PROGRAM Vision
VAR
  trigVisionOk    : R_TRIG;	

//System_Bit
	Always_ON	:	BOOL	:=TRUE	;//상시 ON 
	Always_OFF	:	BOOL	:=FALSE	;//상시 OFF
	
	
	TON_1: TON;
	Time_Data_1: LREAL ;
	
	DATA : LREAL;
	

	CCTV: TON;
	Work_End_Position_Set: BOOL;
	GVL_Vision_ON_Delay_Time: INT;
	test005: BOOL;
	Vision_Delay: BOOL;
	Vision_Delay_TM: TON;
	test01: BOOL;
	Vision_NG_Timer: TON;
	Vision_OFF_Dealy: TON;
	TON_0: TON;
END_VAR
VAR // added by the converter: edge detectors and wires of the graphical bodies
    _rt1, _rt2, _rt3, _rt4, _rt5 : R_TRIG;
    _w1, _w2 : BOOL;
END_VAR

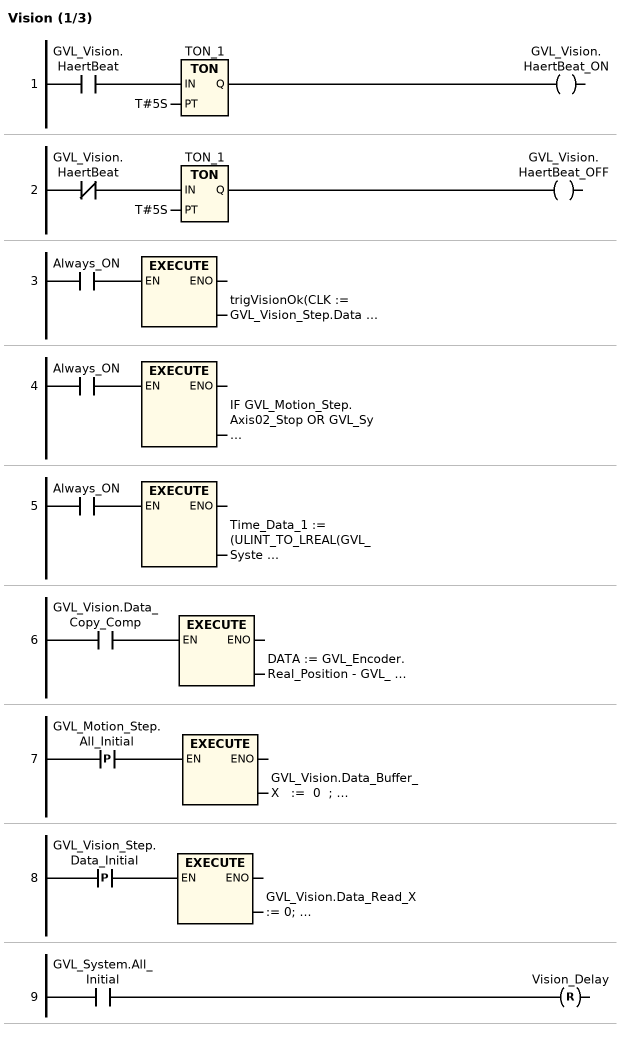
// NETWORK 1
TON_1(IN := GVL_Vision.HaertBeat, PT := T#5S); // TON
GVL_Vision.HaertBeat_ON := TON_1.Q;

// NETWORK 2
TON_1(IN := NOT GVL_Vision.HaertBeat, PT := T#5S); // TON
GVL_Vision.HaertBeat_OFF := TON_1.Q;

// NETWORK 3
IF Always_ON THEN
    trigVisionOk(CLK := GVL_Vision_Step.Data_Initial);
    
    IF trigVisionOk.Q OR GVL_System.All_Initial THEN
    	GVL_Vision.Data_Read_X	:=	0;
    	GVL_Vision.Data_Read_Y	:=	0;
    	GVL_Vision.Data_Read_R	:=	0;
    	GVL_Vision.Vision_OK	:=	FALSE;
    	GVL_Vision.Vision_NG	:=	FALSE;
    END_IF
END_IF

// NETWORK 4
IF Always_ON THEN
    IF GVL_Motion_Step.Axis02_Stop OR GVL_System.All_Initial THEN
    	GVL_Vision.Average_Speed := 0;
    	GVL_Vision.TotalSpeed := 0;
    	GVL_Vision.FrameCount := 0;
    	GVL_Vision.Get_Frame := 0;
    	DATA := 0;
    END_IF
END_IF

// NETWORK 5
IF Always_ON THEN
    
    Time_Data_1 := (ULINT_TO_LREAL(GVL_System.Time_Data) * 1E-7);
    
    IF GVL_Vision.Data_Copy_Comp THEN
    	 GVL_Vision.Moving_Time := Time_Data_1 - GVL_Vision.Get_Frame_Time ;
    END_IF
END_IF

// NETWORK 6
IF GVL_Vision.Data_Copy_Comp THEN
    DATA := GVL_Encoder.Real_Position - GVL_Vision.Encoder_DATA01[GVl_Vision.DATA_COUNT];
    GVL_Vision.Target_X_Real_Position_Data := GVL_Vision.Data_Buffer_X - DATA;
END_IF

// NETWORK 7
_rt1(CLK := GVL_Motion_Step.All_Initial);
IF _rt1.Q THEN
    GVL_Vision.Data_Buffer_X 	:=	0	;
    GVL_Vision.Data_Buffer_Y	:=	0	;
    GVL_Vision.Data_Buffer_R	:=	0	;
    GVL_Vision.Data_Copy_Comp	:=	0	;
    GVL_Vision.Get_Frame_Time	:=	0	;
    GVL_Vision.Target_X_Real_Position_Data	:=	0;	
    GVL_Vision.Press_Speed	:=	0;
    GVL_Vision.Travel_Distance	:=	0;
    GVL_Vision.Moving_Time	:= 0;
    Time_Data_1	:= 0;
END_IF

// NETWORK 8
_rt2(CLK := GVL_Vision_Step.Data_Initial);
IF _rt2.Q THEN
    GVL_Vision.Data_Read_X	:= 0;
    GVL_Vision.Data_Read_Y	:= 0;
    GVL_Vision.Data_Read_R	:= 0;
END_IF

// NETWORK 9
Vision_Delay R= GVL_System.All_Initial;

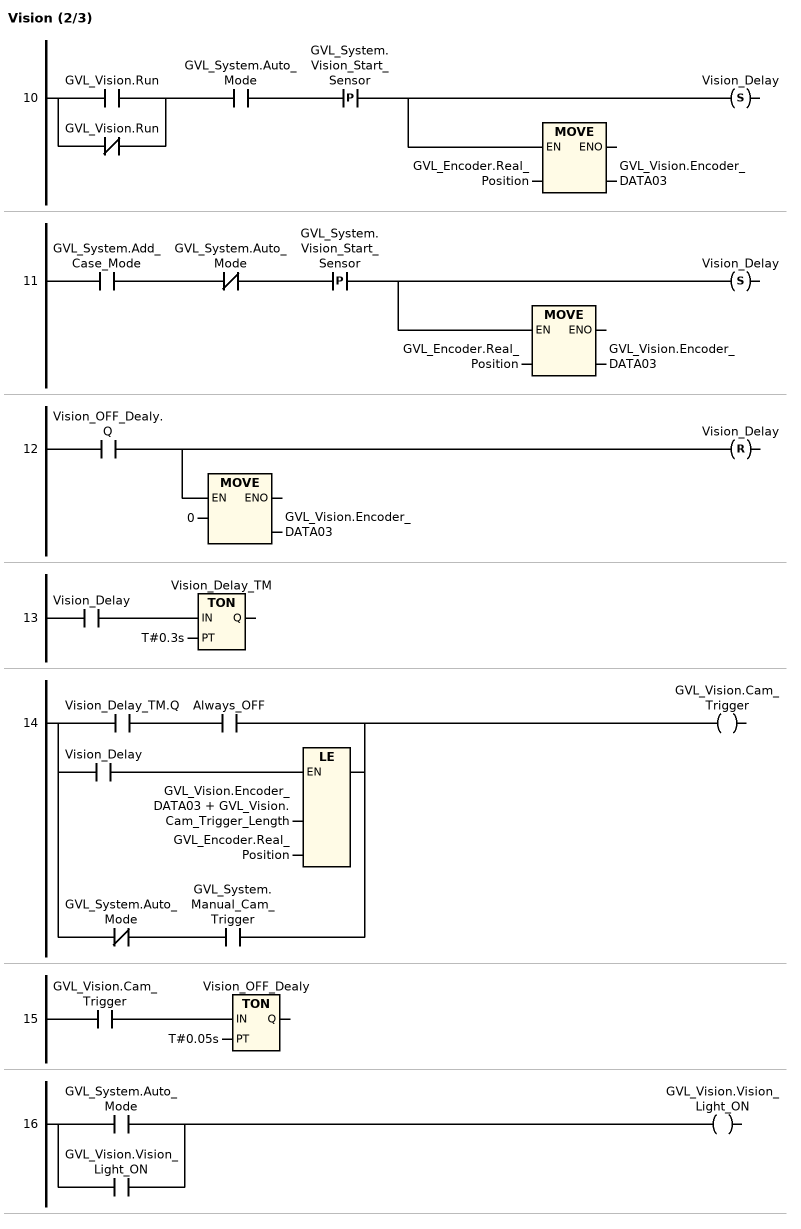
// NETWORK 10
_rt3(CLK := GVL_System.Vision_Start_Sensor);
_w1 := (GVL_Vision.Run OR NOT GVL_Vision.Run) AND GVL_System.Auto_Mode AND _rt3.Q;
Vision_Delay S= _w1;
IF _w1 THEN GVL_Vision.Encoder_DATA03 := GVL_Encoder.Real_Position; END_IF

// NETWORK 11
_rt4(CLK := GVL_System.Vision_Start_Sensor);
_w2 := GVL_System.Add_Case_Mode AND NOT GVL_System.Auto_Mode AND _rt4.Q;
Vision_Delay S= _w2;
IF _w2 THEN GVL_Vision.Encoder_DATA03 := GVL_Encoder.Real_Position; END_IF

// NETWORK 12
Vision_Delay R= Vision_OFF_Dealy.Q;
IF Vision_OFF_Dealy.Q THEN GVL_Vision.Encoder_DATA03 := 0; END_IF

// NETWORK 13
Vision_Delay_TM(IN := Vision_Delay, PT := T#0.3s); // TON

// NETWORK 14
GVL_Vision.Cam_Trigger := Vision_Delay_TM.Q AND Always_OFF OR Vision_Delay AND (GVL_Vision.Encoder_DATA03 + GVL_Vision.Cam_Trigger_Length) <= GVL_Encoder.Real_Position OR NOT GVL_System.Auto_Mode AND GVL_System.Manual_Cam_Trigger;

// NETWORK 15
Vision_OFF_Dealy(IN := GVL_Vision.Cam_Trigger, PT := T#0.05s); // TON

// NETWORK 16
GVL_Vision.Vision_Light_ON := GVL_System.Auto_Mode OR GVL_Vision.Vision_Light_ON;

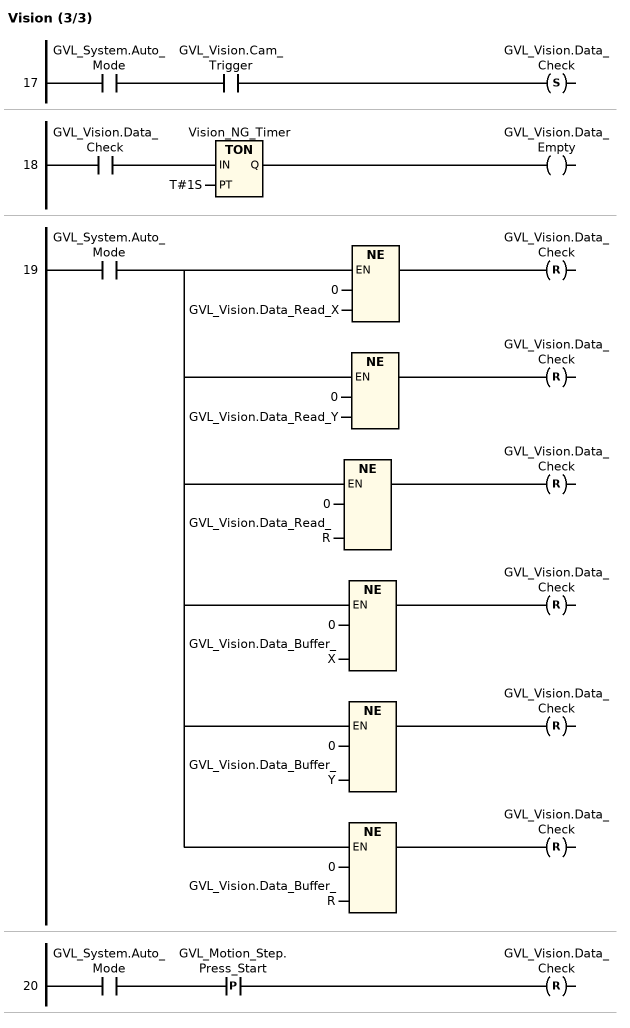
// NETWORK 17
GVL_Vision.Data_Check S= GVL_System.Auto_Mode AND GVL_Vision.Cam_Trigger;

// NETWORK 18
Vision_NG_Timer(IN := GVL_Vision.Data_Check, PT := T#1S); // TON
GVL_Vision.Data_Empty := Vision_NG_Timer.Q;

// NETWORK 19
GVL_Vision.Data_Check R= GVL_System.Auto_Mode AND 0 <> GVL_Vision.Data_Read_X;
GVL_Vision.Data_Check R= GVL_System.Auto_Mode AND 0 <> GVL_Vision.Data_Read_Y;
GVL_Vision.Data_Check R= GVL_System.Auto_Mode AND 0 <> GVL_Vision.Data_Read_R;
GVL_Vision.Data_Check R= GVL_System.Auto_Mode AND 0 <> GVL_Vision.Data_Buffer_X;
GVL_Vision.Data_Check R= GVL_System.Auto_Mode AND 0 <> GVL_Vision.Data_Buffer_Y;
GVL_Vision.Data_Check R= GVL_System.Auto_Mode AND 0 <> GVL_Vision.Data_Buffer_R;

// NETWORK 20
_rt5(CLK := GVL_Motion_Step.Press_Start);
GVL_Vision.Data_Check R= GVL_System.Auto_Mode AND _rt5.Q;

END_PROGRAM

(* stored: Version 1.1.0.1, ProductVersion 3.1.4024.15
   POU Vision: Id {fe608fbf-4e51-40b4-97c4-03055456ca77}, SpecialFunc None *)
